DATA_BLOCK "Process_DB"
{ S7_Optimized_Access := 'TRUE' }
"Process"


BEGIN

END_DATA_BLOCK
